// TIA Portal V19 export
DATA_BLOCK "Filler_CIP_512_DB"   // DB96
{ S7_Optimized_Access := 'TRUE' }
// stored: AutoNumber false, MemoryReserve 0
   VAR RETAIN
      Count : Int;   // Continue cip until count value greater than setpoint in code
      Drain_Ready : Bool;
      M0139_db96 : Bool;   // intermediate bit
      LyeRequest_db96 : Bool;   // intermediate bit
      AcidReques_db96 : Bool;   // intermediate bit
      RequestOffDelay : Bool;   // Request off delay bit
      CIPScreenCenterMessage : Int;
      CIPheld : Bool;
      resumeButton : Bool;
   END_VAR
BEGIN
END_DATA_BLOCK
